Fanuc KAREL source: IO_CLR.kl

--* coding: Shift-jis *--
--
--  --------------------------------------
--  Released under the Apache 2.0 License.
--  Yuki Meguro
--  --------------------------------------
--
--  --------------------------------------
--  Author: Yuki Meguro
--
--  Description:
--    Template Karel File
--
--  Dependancies: none
--  --------------------------------------

PROGRAM IO_CLR
%ALPHABETIZE
%NOLOCKGROUP
%SYSTEM
%NOPAUSESHFT
%NOPAUSE=ERROR+COMMAND+TPENABLE
%ENVIRONMENT REGOPE
%COMMENT='Clear IO'

CONST
null = 17042
err_abort = 2

VAR
status: INTEGER
get_stat: ARRAY[3] OF INTEGER
data_type: INTEGER
data_box: ARRAY[3] OF INTEGER
i: INTEGER
get_int: ARRAY[3] OF INTEGER
get_real: ARRAY[3] OF REAL
get_str: ARRAY[3] OF STRING[30]
exit_loop: BOOLEAN
exit_sloop: BOOLEAN
cin: INTEGER

BEGIN

FOR i = 1 TO 3 DO
	GET_TPE_PRM(i, data_type, get_int[i], get_real[i], get_str[i], get_stat[i])
	IF i < 3 THEN
		IF (get_int[i] < 1) AND (get_stat[i] = 0) THEN
			WRITE(CHR(137),CHR(128))
			WRITE('PRM [', i, ' ]  < 1', CR, '**Value Err**', CR)
			FORCE_SPMENU(TP_PANEL,SPI_TPUSER,1)
			POST_ERR(status, '', 0, err_abort)
		ENDIF
	ENDIF
	IF (get_stat[i] = 0) AND (data_type <> 1) THEN
			WRITE(CHR(137),CHR(128))
			WRITE('PRM [', i, ' ]  Variable Err.', CR, '**Program Stop**', CR)
			FORCE_SPMENU(TP_PANEL,SPI_TPUSER,1)
			POST_ERR(status, '', 0, err_abort)
	ENDIF
	IF i = 2 THEN
		IF (get_stat[1] = 0) AND (get_stat[2] = null) THEN
			WRITE(CHR(137),CHR(128))
			WRITE('PRM [ 2 ]  = null', CR, '**Program Stop**', CR)
			FORCE_SPMENU(TP_PANEL,SPI_TPUSER,1)
			POST_ERR(status, '', 0, err_abort)
		ENDIF
	ENDIF
ENDFOR

IF get_stat[1] = null THEN
		exit_loop = FALSE
		REPEAT
	    WRITE(CHR(137),CHR(128))
			FORCE_SPMENU(TP_PANEL,SPI_TPUSER,1)
			WRITE('===IO CLEAR===', CR)
			WRITE('Please select mode.', CR)
			WRITE('DOUT:0, ROUT:1, END:other', CR)
			READ(get_int[3])

			SELECT get_int[3] OF
				CASE(0):
					WRITE('Clear DOUT mode.', CR)
				CASE(1):
					WRITE('Clear ROUT mode.', CR)
				ELSE:
					WRITE('**Program Stop**', CR)
					ABORT
			ENDSELECT

			exit_sloop = FALSE
			REPEAT
				WRITE('Start IO number', CR)
				READ(get_int[1])
				WRITE('Stop IO number', CR)
				READ(get_int[2])
				IF get_int[1] > get_int[2] THEN
					WRITE('**Value Err**', CR)
				ELSE
					exit_sloop = TRUE
				ENDIF
			UNTIL exit_sloop

			IF get_int[3] = 0 THEN
				WRITE(CR, 'DOUT' , get_int[1] , ' -' , get_int[2] , ' Clear', CR)
			ELSE
				WRITE(CR, 'ROUT' , get_int[1] , ' -' , get_int[2] , ' Clear', CR)
			ENDIF
			WRITE('OK? (YES:0, NO:1, Abort:other)', CR)
			READ(cin)
			SELECT cin OF
				CASE(0):
					exit_loop = TRUE
				CASE(1):
					exit_loop = FALSE
				ELSE:
					exit_loop = TRUE
					cin = 4
			ENDSELECT
			UNTIL exit_loop
ENDIF

IF cin = 4 THEN
	WRITE('**Program Stop**', CR)
	ABORT
ELSE
	IF get_int[3] = 0 THEN
		FOR i = get_int[1] TO get_int[2] DO
			DOUT[i] = OFF
		ENDFOR
		ELSE IF get_int[3] = 1 THEN
			FOR i = get_int[1] TO get_int[2] DO
				RDO[i] = OFF
			ENDFOR
		ENDIF
	ENDIF
ENDIF
END IO_CLR
